// TIA Portal V16 export
// export: Created 2020-03-15T18:15:54.9366545Z, ExportSetting WithDefaults, WithReadOnly, DisplayName Totally Integrated Automation Portal, DisplayVersion V16, DisplayName TIA Portal Version Control Interface, DisplayVersion V16, DisplayName TIA Portal Openness, DisplayVersion V16, DisplayName STEP 7 Professional, DisplayVersion V16, DisplayName STEP 7 Safety, DisplayVersion V16, DisplayName WinCC Advanced, DisplayVersion V16
TYPE "StepValues"
// stored: CreationDate 2020-03-15T17:46:50.1549602Z, InterfaceModifiedDate 2020-03-15T18:09:20.7956673Z, IsConsistent true, IsFailsafeCompliant false, IsKnowHowProtected false, LibraryConformanceStatus Das Objekt ist bibliothekskonform., ModifiedDate 2020-03-15T18:09:26.7487262Z
   STRUCT
      StepMode : Int;   // 0 = Automatic / 1 = SingleStep
      SingleStep : Bool;   // Step once
      CurrentStep : Int;   // Actual step no
      CurrentTime : DInt;   // Actual step time
      CylcleState : Int;   // 1 = running
      CycleAbort : Bool;   // abort cycle
   END_STRUCT;
END_TYPE
